(* CoDeSys 2.3.9.25 project: doma_prazdny.pro *)
(* Libraries: Standard.lib 22.11.04 11:21:12, SYSLIBCALLBACK.LIB 20.4.05 11:04:48 *)

(* PLC configuration (modules and I/O channels)
0750-0502 2 DO 24V DC 2.0A [Type_10_2_Channels] node 0, in %IB0 out %QB0 {INTTypePAAssignment = PLC; INTTypeModule = plugged}
  vstup1 AT %QX4.0 [BOOLOnX_Q] O 1: Digital Output
  vstup2 AT %QX4.1 [BOOLOnX_Q] O 2: Digital Output
0750-0530 8 DO 24 V DC 0.5A [Type_10_8_Channels] node 1, in %IB1 out %QB1 {INTTypePAAssignment = PLC; INTTypeModule = plugged}
  vstup3 AT %QX4.2 [BOOLOnX_Q] O 1: Digital Output
  vstup4 AT %QX4.3 [BOOLOnX_Q] O 2: Digital Output
  AT %QX4.4 [BOOLOnX_Q] O 3: Digital Output
  AT %QX4.5 [BOOLOnX_Q] O 4: Digital Output
  AT %QX4.6 [BOOLOnX_Q] O 5: Digital Output
  AT %QX4.7 [BOOLOnX_Q] O 6: Digital Output
  AT %QX4.8 [BOOLOnX_Q] O 7: Digital Output
  AT %QX4.9 [BOOLOnX_Q] O 8: Digital Output
0750-0530 8 DO 24 V DC 0.5A [Type_10_8_Channels] node 2, in %IB2 out %QB2 {INTTypePAAssignment = PLC; INTTypeModule = plugged}
  AT %QX4.10 [BOOLOnX_Q] O 1: Digital Output
  AT %QX4.11 [BOOLOnX_Q] O 2: Digital Output
  AT %QX4.12 [BOOLOnX_Q] O 3: Digital Output
  AT %QX4.13 [BOOLOnX_Q] O 4: Digital Output
  AT %QX4.14 [BOOLOnX_Q] O 5: Digital Output
  AT %QX4.15 [BOOLOnX_Q] O 6: Digital Output
  AT %QX5.0 [BOOLOnX_Q] O 7: Digital Output
  AT %QX5.1 [BOOLOnX_Q] O 8: Digital Output
0750-0430 8 DI 24 V DC 3.0ms [Type_1_8_Channels] node 3, in %IB3 out %QB3 {INTTypePAAssignment = PLC; INTTypeModule = plugged}
  AT %IX8.0 [BOOLOnX_I] I 1: Digital Input
  AT %IX8.1 [BOOLOnX_I] I 2: Digital Input
  AT %IX8.2 [BOOLOnX_I] I 3: Digital Input
  AT %IX8.3 [BOOLOnX_I] I 4: Digital Input
  AT %IX8.4 [BOOLOnX_I] I 5: Digital Input
  AT %IX8.5 [BOOLOnX_I] I 6: Digital Input
  AT %IX8.6 [BOOLOnX_I] I 7: Digital Input
  AT %IX8.7 [BOOLOnX_I] I 8: Digital Input
0750-0430 8 DI 24 V DC 3.0ms [Type_1_8_Channels] node 4, in %IB4 out %QB4 {INTTypePAAssignment = PLC; INTTypeModule = plugged}
  AT %IX8.8 [BOOLOnX_I] I 1: Digital Input
  AT %IX8.9 [BOOLOnX_I] I 2: Digital Input
  AT %IX8.10 [BOOLOnX_I] I 3: Digital Input
  AT %IX8.11 [BOOLOnX_I] I 4: Digital Input
  AT %IX8.12 [BOOLOnX_I] I 5: Digital Input
  AT %IX8.13 [BOOLOnX_I] I 6: Digital Input
  AT %IX8.14 [BOOLOnX_I] I 7: Digital Input
  AT %IX8.15 [BOOLOnX_I] I 8: Digital Input
0750-0464#04 2/4 AI RTD / ADJ./ HA [Type_44_4_Channels] node 5, in %IB5 out %QB5 {INTTypePAAssignment = PLC; INTTypeModule = plugged}
  AT %IW0 [INTOnW_I] Channel 1
  AT %IW1 [INTOnW_I] Channel 2
  AT %IW2 [INTOnW_I] Channel 3
  AT %IW3 [INTOnW_I] Channel 4
0750-0559 4 AO 0-10V DC [Type_14_4_Channels] node 6, in %IB6 out %QB6 {INTTypePAAssignment = PLC; INTTypeModule = plugged}
  AT %QW0 [WORDOnW_Q] O 1: Analog Output
  AT %QW1 [WORDOnW_Q] O 2: Analog Output
  AT %QW2 [WORDOnW_Q] O 3: Analog Output
  AT %QW3 [WORDOnW_Q] O 4: Analog Output
0750-0455 4 AI 4-20mA s.e. [Type_8_4_Channels] node 7, in %IB7 out %QB7 {INTTypePAAssignment = PLC; INTTypeModule = plugged}
  AT %IW4 [WORDOnW_I] I 1: Analog Input
  AT %IW5 [WORDOnW_I] I 2: Analog Input
  AT %IW6 [WORDOnW_I] I 3: Analog Input
  AT %IW7 [WORDOnW_I] I 4: Analog Input
Fieldbus variables [FB_VARS] node 1, in %IB0 out %QB0
*)

(* POU PLC_PRG, LD *)
PROGRAM PLC_PRG
VAR
END_VAR
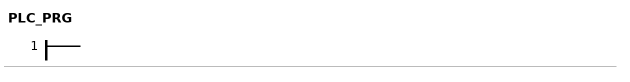
_LD_ (* Ladder Diagram *)
NETWORK 1
	*
_END_LD_
(* the same logic as Structured Text *)
(* Network 1 *)
END_PROGRAM
